Staubli VAL3: SaveNewProduct.pgx

public program SaveNewProduct(bool& x_bRes (dimensions=1))
  local num l_nTrajIndex
  local string l_sFileName
  local string l_sSBuff
begin

  //建立生产文件头的文件头


  //参数初始化
  x_bRes=false
  l_sFileName="Disk://Txt/Recipe.txt"

  //××××××××××××××××××××××××××××××××××××××××××××××××××××××××××××××××××××
  //开始部分
  //关闭所有文件
  call FileDir:CloseAllFile()

  //文件是否可以打开
  nFileID=$fileOpen(l_sFileName,"w")
  if nFileID<0 or nFileID>9
    return
  endIf

  //工具
  l_sSBuff="PRODUCT=TEST"
  if $fileSet(nFileID,l_sSBuff,1)!=1
    return
  endIf


  //工具
  l_sSBuff="TOOL="
  l_sSBuff=l_sSBuff+toString(".3",tCfg.trsf.x)+","+toString(".3",tCfg.trsf.y)+","+toString(".3",tCfg.trsf.z)+","
  l_sSBuff=l_sSBuff+toString(".3",tCfg.trsf.rx)+","+toString(".3",tCfg.trsf.ry)+","+toString(".3",tCfg.trsf.rz)
  if $fileSet(nFileID,l_sSBuff,1)!=1
    return
  endIf

  l_sSBuff="TOTALELEMENTS=0"
  if $fileSet(nFileID,l_sSBuff,1)!=1
    return
  endIf

  l_sSBuff="FRAME=0,0,0,0,0,0"
  if $fileSet(nFileID,l_sSBuff,1)!=1
    return
  endIf

  l_sSBuff="OFFSET=0,0,0,0,0,0"
  if $fileSet(nFileID,l_sSBuff,1)!=1
    return
  endIf

  l_sSBuff="PRESET=StaubliPreset"
  if $fileSet(nFileID,l_sSBuff,1)!=1
    return
  endIf

  l_sSBuff=""
  if $fileSet(nFileID,l_sSBuff,1)!=1
    return
  endIf

  l_sSBuff=""
  if $fileSet(nFileID,l_sSBuff,1)!=1
    return
  endIf

  //××××××××××××××××××××××××××××××××××××××××××××××××××××××××××××××××××
  //重命名
  //关闭所有文件
  call FileDir:CloseAllFile()

  x_bRes=true

end
